# EPICS substitutions: ek9000App/Db/EL2042.substitutions
file EL2042.template
{       pattern
        {
                TERMINAL,

        }
        {
        }
}
